// TIA Portal V20 export
DATA_BLOCK "RecipeParameter"   // DB115
// stored: Access Published, MemoryReserve 100
   VAR
      SelectdRecipeTypeID : Int;
      SelectdRecipeID : Int;
      CurrentRecipeName : WString;
      CurrentRecipeID : Int;
      GetParameterSetName : Int;
      ParametersSV : "HMI_IF_Parameter_ListRecipe_UDT";
      ParametersPV : "HMI_IF_Parameter_ListRecipe_UDT";
   END_VAR
BEGIN
END_DATA_BLOCK
